// TIA Portal project "ArtecPLC" (V15)

(* hardware
DEVICE "S71500/ET200MP station_1"  S7-1500 station
   slot 0: "Telaio di montaggio_0"  Rack  6ES7 590-1***0-0AA0
   slot 1: "Stazione Principale"  CPU 1515-2 PN  6ES7 515-2AM01-0AB0  V2.5
      slot 3: "Display CPU_1"  6ES7591-1BA00-0AA0
*)

// ===== PLC "Stazione Principale"  CPU 1515-2 PN =====

DATA_BLOCK "DosatoreManuale_DB"   // DB4
{ S7_Optimized_Access := 'TRUE' }
AUTHOR : Valentino-Fabbri
VERSION : 1.14
// stored: InstanceOfName DosatoreManuale
"DosatoreManuale"
BEGIN
END_DATA_BLOCK

// folder: System blocks/Program resources

DATA_BLOCK "ImpulsoEVGas_FB_DosatoreManuale"   // DB1
{ S7_Optimized_Access := 'TRUE' }
AUTHOR : Simatic
FAMILY : IEC
NAME : IEC_TMR
VERSION : 1.0
// stored: InstanceOfName IEC_TIMER
"IEC_TIMER"
BEGIN
END_DATA_BLOCK

DATA_BLOCK "ImpulsoMixer_GasPresente_FB_DosatoreManuale"   // DB2
{ S7_Optimized_Access := 'TRUE' }
AUTHOR : Simatic
FAMILY : IEC
NAME : IEC_TMR
VERSION : 1.0
// stored: InstanceOfName IEC_TIMER
"IEC_TIMER"
BEGIN
END_DATA_BLOCK

DATA_BLOCK "ImpulsoDisco_FB_DosatoreManuale"   // DB3
{ S7_Optimized_Access := 'TRUE' }
AUTHOR : Simatic
FAMILY : IEC
NAME : IEC_TMR
VERSION : 1.0
// stored: InstanceOfName IEC_TIMER
"IEC_TIMER"
BEGIN
END_DATA_BLOCK

// folder: (top level)

FUNCTION_BLOCK "DosatoreManuale"   // FB1, LAD
TITLE = Blocco Dosatore in Manuale
{ S7_Optimized_Access := 'TRUE' }
AUTHOR : Valentino-Fabbri
VERSION : 1.14
   VAR_INPUT
      StopEmergenza : Bool;   // Fornire un bit che se aperto fermi tutto
      GasInPressione : Bool;   // Bit che mi fornisce lo stato del Gas In Pressione
      GasARegime : Bool;   // Bit che mi fornisce lo stato del Gas a Regime
      GasAZero : Bool;   // Bit che mi fornisce lo stato del Gas a zero
      DiscoARegime : Bool;   // Bit che mi fornisce lo stato del Disco a Regime
      DiscoAZero : Bool;   // Bit che mi fornisce lo stato del Disco a zero
      MixerARegime : Bool;   // Bit che mi fornisce lo stato del mixer a Regime
      MixerAZero : Bool;   // Bit che mi fornisce lo stato del mixer a Zero
      DosatoriOkInRicetta : Bool;   // Bit che mi indica se i dosatori sono presenti ed in ricetta
      RicettaMixer : Real;   // Valore fornito dal cliente - misurato in RPM
      RicettaDisco : Real;   // Valore fornito dal cliente - misurato in RPM
      RicettaGas : Real;   // Valore fornito dal cliente - misurato in LPM
      TipoDiAvvio : Bool;   // Modalità di avvio Disco - se prima Disco e poi Mixer, oppure Mixer e poi Disco
   END_VAR
   VAR_OUTPUT
      EVGas : Bool;   // Elettrovalvola Gas Argon
      Mixer : Bool;   // Abilitazione Mixer
      Disco : Bool;   // Abilitazione Disco
      DosatoreAcceso : Bool;   // Flag che indica il dosatore a Regime
   END_VAR
   VAR_IN_OUT
      PulsanteMixerHMI : Bool;   // Pulsante Mixer da HMI
      PulsanteDiscoHMI : Bool;   // Pulsante Disco da HMI
      PulsanteGasHMI : Bool;   // Pulsante Gas da HMI
      PulsanteStopMixer : Bool;   // Stop Mixer da HMI
      PulsanteStopDisco : Bool;   // Stop Disco da HMI
      PulsanteStopGas : Bool;   // Stop Gas da HMI
      ValoreComandoMixer : Real;   // Valore di comando velocità Mixer
      ValoreComandoDisco : Real;   // Valore di comando velocità Disco
      ValoreComandoGas : Real;   // Valore di comando flusso Gas
   END_VAR
   VAR_TEMP
      CondizioniRispettate : Bool;
      "Step" : Array[1..10] of Bool;
      DosatoreSpento : Bool;
      AppoggioPulsanteGas : Bool;
      AppoggioPulsanteMixer : Bool;
      AppoggioPulsanteDisco : Bool;
      AppoggioStopGasDaMixerODisco : Bool;
      AppoggioStopMixerDaDisco : Bool;
      AppoggioStopDiscoDaMixer : Bool;
      StopGas : Bool;
      StopDisco : Bool;
      StopMixer : Bool;
   END_VAR
   VAR_TEMP   // added for the SCL form of the ladder/FBD networks
      _w1 : Bool;
      _w2 : Bool;
      _w3 : Bool;
      _w4 : Bool;
      _w5 : Bool;
      _w6 : Bool;
      _w7 : Bool;
      _w8 : Bool;
      _w9 : Bool;
      _w10 : Bool;
      _w11 : Bool;
      _w12 : Bool;
      _w13 : Bool;
      _w14 : Bool;
   END_VAR
BEGIN

REGION Network 1: Condizioni Iniziali
   // Lo stop di emergenza è un bit che normalmente è chiuso e se aperto vuoldire che una condizione è venuta a mancare in cabina
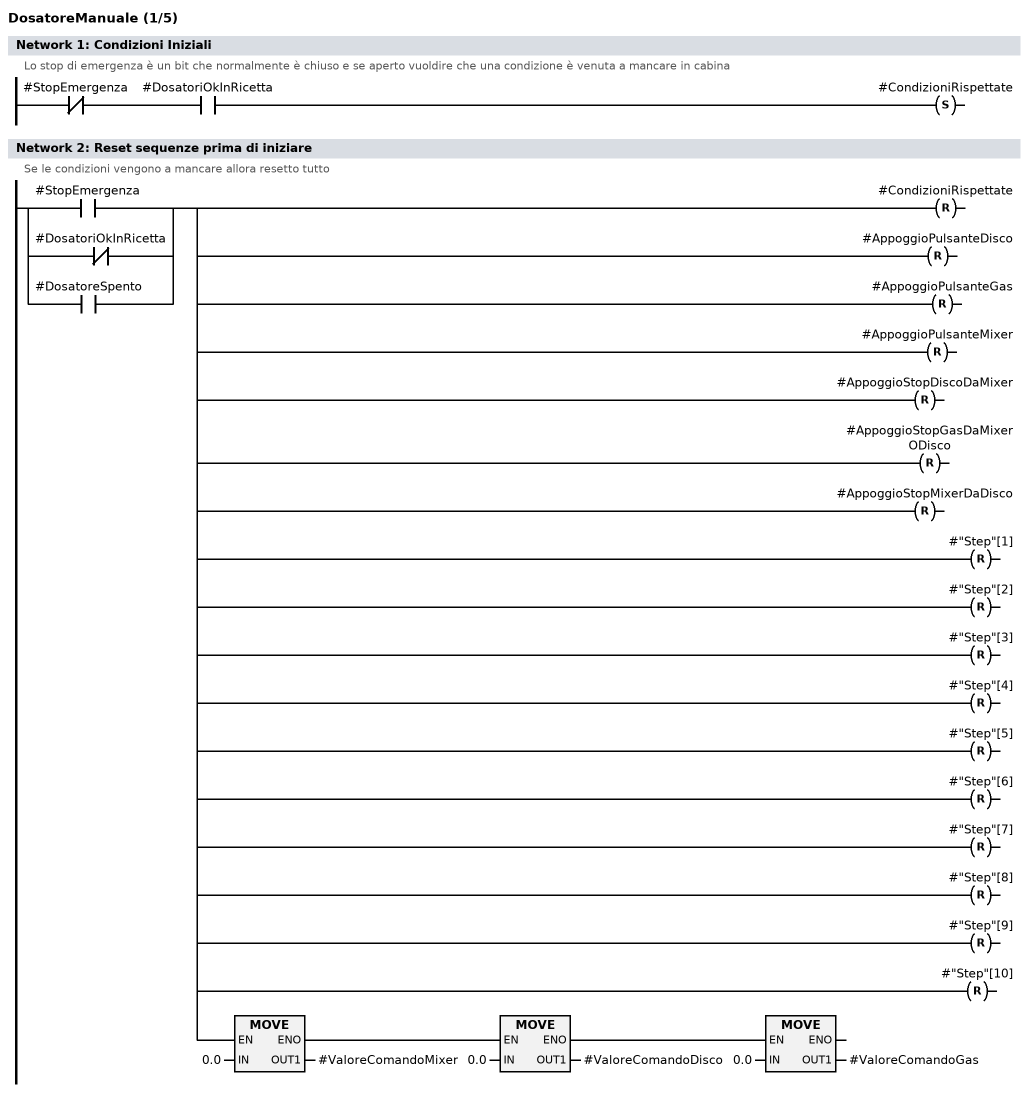
   RUNG wire#powerrail
      I_Contact( #StopEmergenza )
      Contact( #DosatoriOkInRicetta )
      S_Coil( #CondizioniRispettate )
   END_RUNG
   // the same network as SCL:
   IF NOT #StopEmergenza AND #DosatoriOkInRicetta THEN #CondizioniRispettate := TRUE; END_IF;
END_REGION

REGION Network 2: Reset sequenze prima di iniziare
   // Se le condizioni vengono a mancare allora resetto tutto
   RUNG wire#powerrail
      Contact( #StopEmergenza )
      wire#w1
      R_Coil( #CondizioniRispettate )
   END_RUNG
   RUNG wire#powerrail
      I_Contact( #DosatoriOkInRicetta )
   END_RUNG wire#w1
   RUNG wire#powerrail
      Contact( #DosatoreSpento )
   END_RUNG wire#w1
   RUNG wire#w1
      R_Coil( #AppoggioPulsanteDisco )
   END_RUNG
   RUNG wire#w1
      R_Coil( #AppoggioPulsanteGas )
   END_RUNG
   RUNG wire#w1
      R_Coil( #AppoggioPulsanteMixer )
   END_RUNG
   RUNG wire#w1
      R_Coil( #AppoggioStopDiscoDaMixer )
   END_RUNG
   RUNG wire#w1
      R_Coil( #AppoggioStopGasDaMixerODisco )
   END_RUNG
   RUNG wire#w1
      R_Coil( #AppoggioStopMixerDaDisco )
   END_RUNG
   RUNG wire#w1
      R_Coil( #"Step"[1] )
   END_RUNG
   RUNG wire#w1
      R_Coil( #"Step"[2] )
   END_RUNG
   RUNG wire#w1
      R_Coil( #"Step"[3] )
   END_RUNG
   RUNG wire#w1
      R_Coil( #"Step"[4] )
   END_RUNG
   RUNG wire#w1
      R_Coil( #"Step"[5] )
   END_RUNG
   RUNG wire#w1
      R_Coil( #"Step"[6] )
   END_RUNG
   RUNG wire#w1
      R_Coil( #"Step"[7] )
   END_RUNG
   RUNG wire#w1
      R_Coil( #"Step"[8] )
   END_RUNG
   RUNG wire#w1
      R_Coil( #"Step"[9] )
   END_RUNG
   RUNG wire#w1
      R_Coil( #"Step"[10] )
   END_RUNG
   RUNG wire#w1
      Move(in := 0.0, out1 => #ValoreComandoMixer)
      Move(in := 0.0, out1 => #ValoreComandoDisco)
      Move(in := 0.0, out1 => #ValoreComandoGas)
   END_RUNG
   // the same network as SCL:
   IF #StopEmergenza OR NOT #DosatoriOkInRicetta OR #DosatoreSpento THEN
       #CondizioniRispettate := FALSE;
       #AppoggioPulsanteDisco := FALSE;
       #AppoggioPulsanteGas := FALSE;
       #AppoggioPulsanteMixer := FALSE;
       #AppoggioStopDiscoDaMixer := FALSE;
       #AppoggioStopGasDaMixerODisco := FALSE;
       #AppoggioStopMixerDaDisco := FALSE;
       #"Step"[1] := FALSE;
       #"Step"[2] := FALSE;
       #"Step"[3] := FALSE;
       #"Step"[4] := FALSE;
       #"Step"[5] := FALSE;
       #"Step"[6] := FALSE;
       #"Step"[7] := FALSE;
       #"Step"[8] := FALSE;
       #"Step"[9] := FALSE;
       #"Step"[10] := FALSE;
       #ValoreComandoMixer := 0.0;
       #ValoreComandoDisco := 0.0;
       #ValoreComandoGas := 0.0;
   END_IF;
END_REGION

REGION Network 3: Pulsanti di Stop
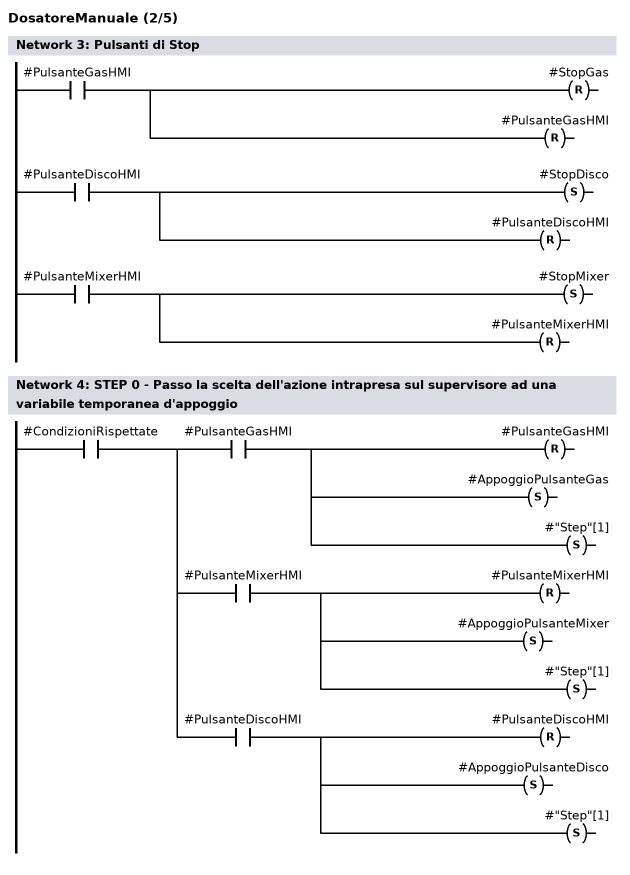
   RUNG wire#powerrail
      Contact( #PulsanteGasHMI )
      wire#w1
      R_Coil( #StopGas )
   END_RUNG
   RUNG wire#w1
      R_Coil( #PulsanteGasHMI )
   END_RUNG
   RUNG wire#powerrail
      Contact( #PulsanteDiscoHMI )
      wire#w2
      S_Coil( #StopDisco )
   END_RUNG
   RUNG wire#w2
      R_Coil( #PulsanteDiscoHMI )
   END_RUNG
   RUNG wire#powerrail
      Contact( #PulsanteMixerHMI )
      wire#w3
      S_Coil( #StopMixer )
   END_RUNG
   RUNG wire#w3
      R_Coil( #PulsanteMixerHMI )
   END_RUNG
   // the same network as SCL:
   IF #PulsanteGasHMI THEN
       #StopGas := FALSE;
       #PulsanteGasHMI := FALSE;
   END_IF;
   IF #PulsanteDiscoHMI THEN
       #StopDisco := TRUE;
       #PulsanteDiscoHMI := FALSE;
   END_IF;
   IF #PulsanteMixerHMI THEN
       #StopMixer := TRUE;
       #PulsanteMixerHMI := FALSE;
   END_IF;
END_REGION

REGION Network 4: STEP 0 - Passo la scelta dell'azione intrapresa sul supervisore ad una variabile temporanea d'appoggio
   RUNG wire#powerrail
      Contact( #CondizioniRispettate )
      wire#w1
      Contact( #PulsanteGasHMI )
      wire#w2
      R_Coil( #PulsanteGasHMI )
   END_RUNG
   RUNG wire#w2
      S_Coil( #AppoggioPulsanteGas )
   END_RUNG
   RUNG wire#w2
      S_Coil( #"Step"[1] )
   END_RUNG
   RUNG wire#w1
      Contact( #PulsanteMixerHMI )
      wire#w3
      R_Coil( #PulsanteMixerHMI )
   END_RUNG
   RUNG wire#w3
      S_Coil( #AppoggioPulsanteMixer )
   END_RUNG
   RUNG wire#w3
      S_Coil( #"Step"[1] )
   END_RUNG
   RUNG wire#w1
      Contact( #PulsanteDiscoHMI )
      wire#w4
      R_Coil( #PulsanteDiscoHMI )
   END_RUNG
   RUNG wire#w4
      S_Coil( #AppoggioPulsanteDisco )
   END_RUNG
   RUNG wire#w4
      S_Coil( #"Step"[1] )
   END_RUNG
   // the same network as SCL:
   #_w1 := #CondizioniRispettate AND #PulsanteGasHMI;
   IF #_w1 THEN
       #PulsanteGasHMI := FALSE;
       #AppoggioPulsanteGas := TRUE;
       #"Step"[1] := TRUE;
   END_IF;
   #_w2 := #CondizioniRispettate AND #PulsanteMixerHMI;
   IF #_w2 THEN
       #PulsanteMixerHMI := FALSE;
       #AppoggioPulsanteMixer := TRUE;
       #"Step"[1] := TRUE;
   END_IF;
   #_w3 := #CondizioniRispettate AND #PulsanteDiscoHMI;
   IF #_w3 THEN
       #PulsanteDiscoHMI := FALSE;
       #AppoggioPulsanteDisco := TRUE;
       #"Step"[1] := TRUE;
   END_IF;
END_REGION

REGION Network 5: STEP 1 - Applico l'azione corrispondente alla scelta effettuata nel segmento precedente
   // Se ho premuto il pulsante GAS - faccio partire solo il GAS
   // Se ho premuto il pulsante Mixer - faccio partire il GAS se non è ancora partito e poi il mixer
   // Se ho premuto il pulsante Disco - faccio partire il GAS , controllo il Tipo Di Avvio, Se Disco-Mixer o Mixer-Disco a seconda di quello partono in rampa il mixer e il disco uno dopo l'altro o viceversa
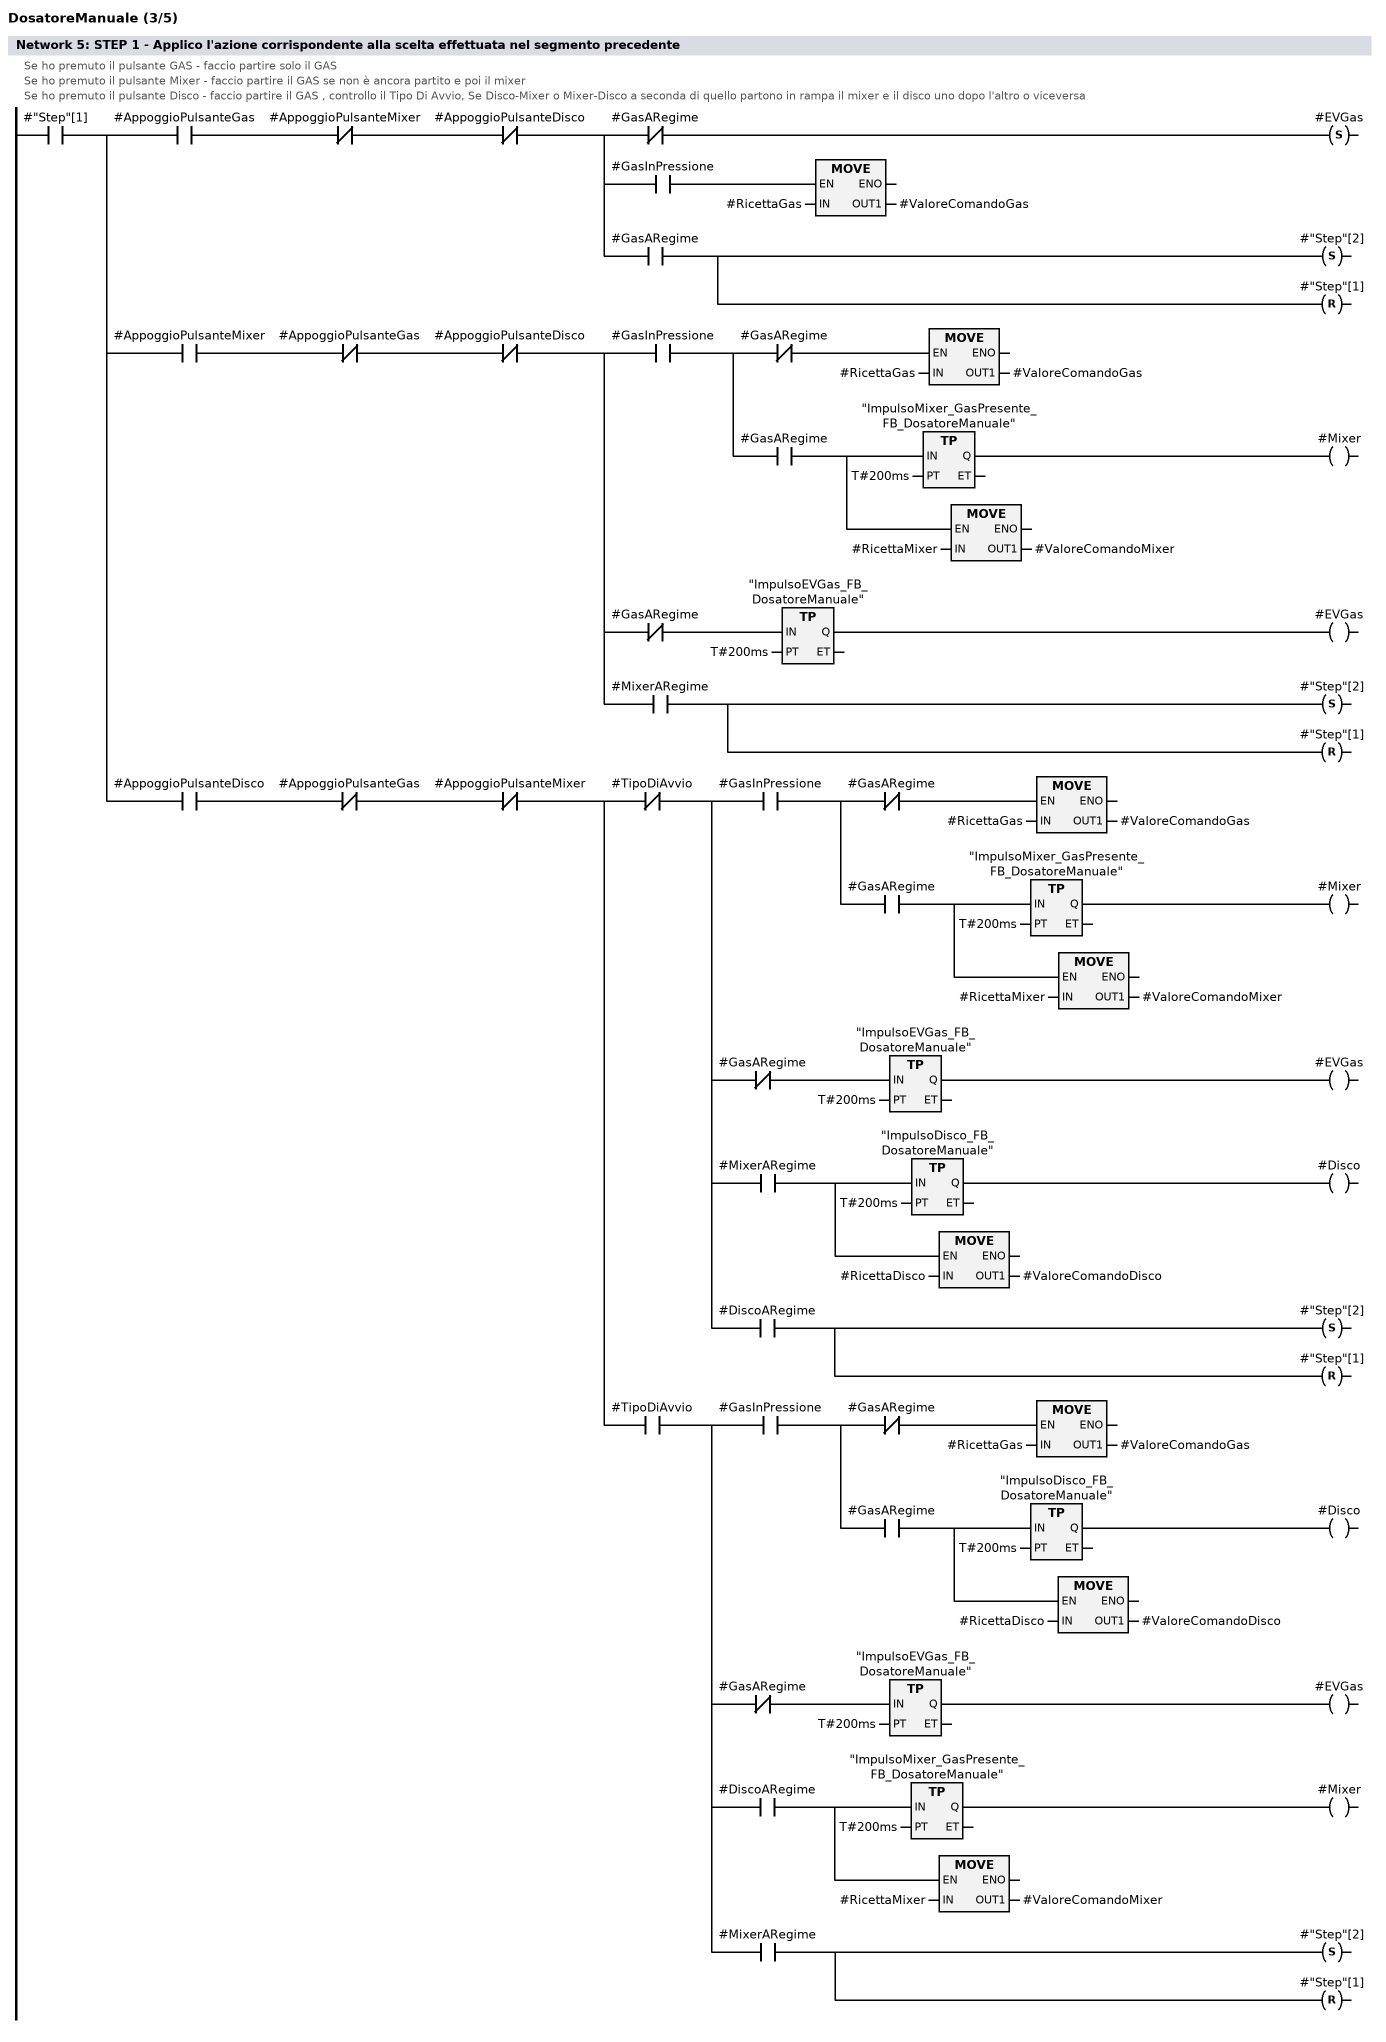
   #_w1 := #"Step"[1] AND #AppoggioPulsanteGas AND NOT #AppoggioPulsanteMixer AND NOT #AppoggioPulsanteDisco;
   IF #_w1 AND NOT #GasARegime THEN #EVGas := TRUE; END_IF;
   IF #_w1 AND #GasInPressione THEN #ValoreComandoGas := #RicettaGas; END_IF;
   #_w2 := #"Step"[1];
   IF #_w1 AND #GasARegime THEN
       #"Step"[2] := TRUE;
       #"Step"[1] := FALSE;
   END_IF;
   #_w3 := #_w2 AND #AppoggioPulsanteMixer AND NOT #AppoggioPulsanteGas AND NOT #AppoggioPulsanteDisco;
   #_w4 := #_w3 AND #GasInPressione;
   IF #_w4 AND NOT #GasARegime THEN #ValoreComandoGas := #RicettaGas; END_IF;
   #_w5 := #_w4 AND #GasARegime;
   "ImpulsoMixer_GasPresente_FB_DosatoreManuale".TP(IN := #_w5, PT := T#200ms);
   #Mixer := "ImpulsoMixer_GasPresente_FB_DosatoreManuale".Q;
   IF #_w5 THEN #ValoreComandoMixer := #RicettaMixer; END_IF;
   "ImpulsoEVGas_FB_DosatoreManuale".TP(IN := #_w3 AND NOT #GasARegime, PT := T#200ms);
   #EVGas := "ImpulsoEVGas_FB_DosatoreManuale".Q;
   IF #_w3 AND #MixerARegime THEN
       #"Step"[2] := TRUE;
       #"Step"[1] := FALSE;
   END_IF;
   #_w6 := #_w2 AND #AppoggioPulsanteDisco AND NOT #AppoggioPulsanteGas AND NOT #AppoggioPulsanteMixer;
   #_w7 := #_w6 AND NOT #TipoDiAvvio;
   #_w8 := #_w7 AND #GasInPressione;
   IF #_w8 AND NOT #GasARegime THEN #ValoreComandoGas := #RicettaGas; END_IF;
   #_w9 := #_w8 AND #GasARegime;
   "ImpulsoMixer_GasPresente_FB_DosatoreManuale".TP(IN := #_w9, PT := T#200ms);
   #Mixer := "ImpulsoMixer_GasPresente_FB_DosatoreManuale".Q;
   IF #_w9 THEN #ValoreComandoMixer := #RicettaMixer; END_IF;
   "ImpulsoEVGas_FB_DosatoreManuale".TP(IN := #_w7 AND NOT #GasARegime, PT := T#200ms);
   #EVGas := "ImpulsoEVGas_FB_DosatoreManuale".Q;
   #_w10 := #_w7 AND #MixerARegime;
   "ImpulsoDisco_FB_DosatoreManuale".TP(IN := #_w10, PT := T#200ms);
   #Disco := "ImpulsoDisco_FB_DosatoreManuale".Q;
   IF #_w10 THEN #ValoreComandoDisco := #RicettaDisco; END_IF;
   IF #_w7 AND #DiscoARegime THEN
       #"Step"[2] := TRUE;
       #"Step"[1] := FALSE;
   END_IF;
   #_w11 := #_w6 AND #TipoDiAvvio;
   #_w12 := #_w11 AND #GasInPressione;
   IF #_w12 AND NOT #GasARegime THEN #ValoreComandoGas := #RicettaGas; END_IF;
   #_w13 := #_w12 AND #GasARegime;
   "ImpulsoDisco_FB_DosatoreManuale".TP(IN := #_w13, PT := T#200ms);
   #Disco := "ImpulsoDisco_FB_DosatoreManuale".Q;
   IF #_w13 THEN #ValoreComandoDisco := #RicettaDisco; END_IF;
   "ImpulsoEVGas_FB_DosatoreManuale".TP(IN := #_w11 AND NOT #GasARegime, PT := T#200ms);
   #EVGas := "ImpulsoEVGas_FB_DosatoreManuale".Q;
   #_w14 := #_w11 AND #DiscoARegime;
   "ImpulsoMixer_GasPresente_FB_DosatoreManuale".TP(IN := #_w14, PT := T#200ms);
   #Mixer := "ImpulsoMixer_GasPresente_FB_DosatoreManuale".Q;
   IF #_w14 THEN #ValoreComandoMixer := #RicettaMixer; END_IF;
   IF #_w11 AND #MixerARegime THEN
       #"Step"[2] := TRUE;
       #"Step"[1] := FALSE;
   END_IF;
END_REGION

REGION Network 6: STEP 2 - Spegnimento Gas o Mixer e poi Gas
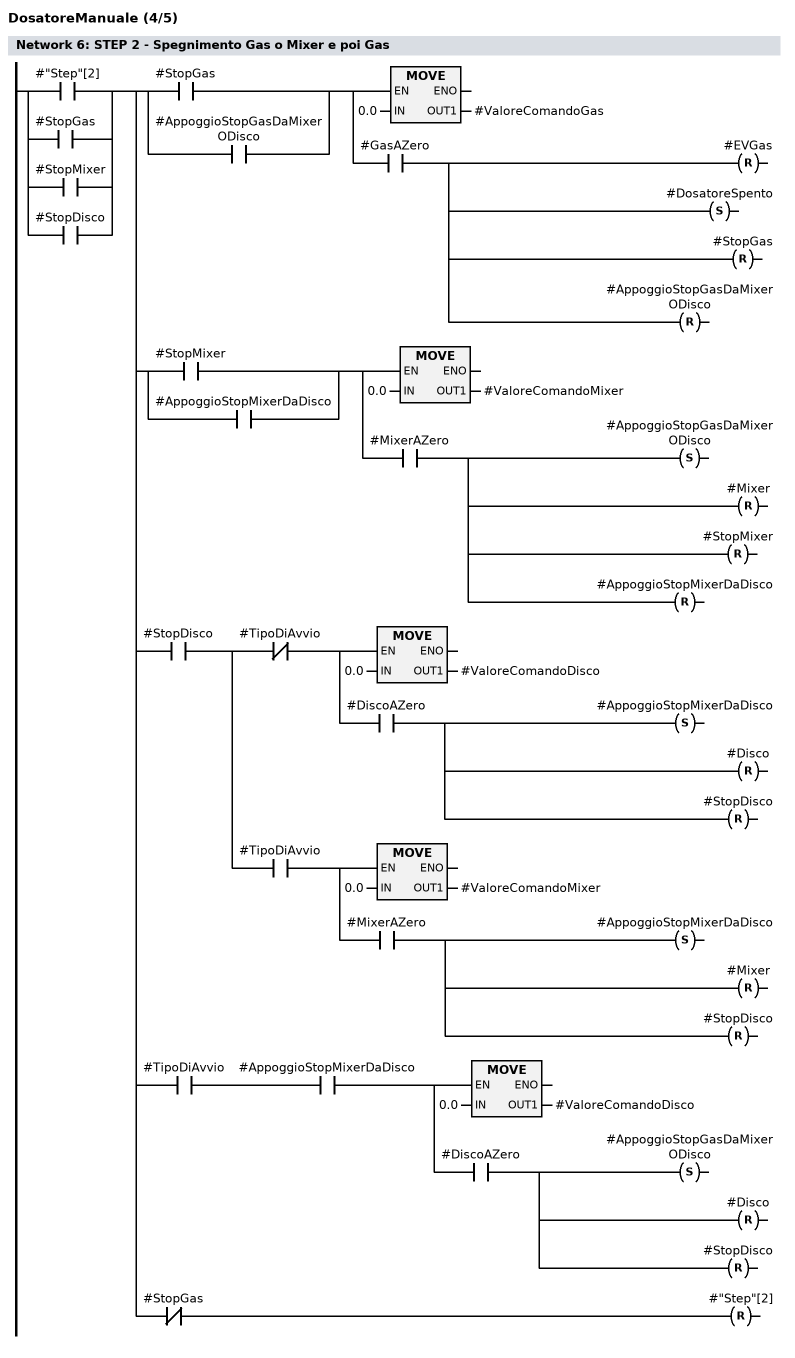
   RUNG wire#powerrail
      Contact( #"Step"[2] )
      wire#w1
      Contact( #StopGas )
      wire#w2
      Move(in := 0.0, out1 => #ValoreComandoGas)
   END_RUNG
   RUNG wire#powerrail
      Contact( #StopGas )
   END_RUNG wire#w1
   RUNG wire#powerrail
      Contact( #StopMixer )
   END_RUNG wire#w1
   RUNG wire#powerrail
      Contact( #StopDisco )
   END_RUNG wire#w1
   RUNG wire#w1
      Contact( #AppoggioStopGasDaMixerODisco )
   END_RUNG wire#w2
   RUNG wire#w2
      Contact( #GasAZero )
      wire#w3
      R_Coil( #EVGas )
   END_RUNG
   RUNG wire#w3
      S_Coil( #DosatoreSpento )
   END_RUNG
   RUNG wire#w3
      R_Coil( #StopGas )
   END_RUNG
   RUNG wire#w3
      R_Coil( #AppoggioStopGasDaMixerODisco )
   END_RUNG
   RUNG wire#w1
      Contact( #StopMixer )
      wire#w4
      Move(in := 0.0, out1 => #ValoreComandoMixer)
   END_RUNG
   RUNG wire#w1
      Contact( #AppoggioStopMixerDaDisco )
   END_RUNG wire#w4
   RUNG wire#w4
      Contact( #MixerAZero )
      wire#w5
      S_Coil( #AppoggioStopGasDaMixerODisco )
   END_RUNG
   RUNG wire#w5
      R_Coil( #Mixer )
   END_RUNG
   RUNG wire#w5
      R_Coil( #StopMixer )
   END_RUNG
   RUNG wire#w5
      R_Coil( #AppoggioStopMixerDaDisco )
   END_RUNG
   RUNG wire#w1
      Contact( #StopDisco )
      wire#w6
      I_Contact( #TipoDiAvvio )
      wire#w7
      Move(in := 0.0, out1 => #ValoreComandoDisco)
   END_RUNG
   RUNG wire#w7
      Contact( #DiscoAZero )
      wire#w8
      S_Coil( #AppoggioStopMixerDaDisco )
   END_RUNG
   RUNG wire#w8
      R_Coil( #Disco )
   END_RUNG
   RUNG wire#w8
      R_Coil( #StopDisco )
   END_RUNG
   RUNG wire#w6
      Contact( #TipoDiAvvio )
      wire#w9
      Move(in := 0.0, out1 => #ValoreComandoMixer)
   END_RUNG
   RUNG wire#w9
      Contact( #MixerAZero )
      wire#w10
      S_Coil( #AppoggioStopMixerDaDisco )
   END_RUNG
   RUNG wire#w10
      R_Coil( #Mixer )
   END_RUNG
   RUNG wire#w10
      R_Coil( #StopDisco )
   END_RUNG
   RUNG wire#w1
      Contact( #TipoDiAvvio )
      Contact( #AppoggioStopMixerDaDisco )
      wire#w11
      Move(in := 0.0, out1 => #ValoreComandoDisco)
   END_RUNG
   RUNG wire#w11
      Contact( #DiscoAZero )
      wire#w12
      S_Coil( #AppoggioStopGasDaMixerODisco )
   END_RUNG
   RUNG wire#w12
      R_Coil( #Disco )
   END_RUNG
   RUNG wire#w12
      R_Coil( #StopDisco )
   END_RUNG
   RUNG wire#w1
      I_Contact( #StopGas )
      R_Coil( #"Step"[2] )
   END_RUNG
   // the same network as SCL:
   #_w1 := #"Step"[2] OR #StopGas OR #StopMixer OR #StopDisco;
   #_w2 := #_w1 AND (#StopGas OR #AppoggioStopGasDaMixerODisco);
   IF #_w2 THEN #ValoreComandoGas := 0.0; END_IF;
   IF #_w2 AND #GasAZero THEN
       #EVGas := FALSE;
       #DosatoreSpento := TRUE;
       #StopGas := FALSE;
       #AppoggioStopGasDaMixerODisco := FALSE;
   END_IF;
   #_w3 := #_w1 AND (#StopMixer OR #AppoggioStopMixerDaDisco);
   IF #_w3 THEN #ValoreComandoMixer := 0.0; END_IF;
   IF #_w3 AND #MixerAZero THEN
       #AppoggioStopGasDaMixerODisco := TRUE;
       #Mixer := FALSE;
       #StopMixer := FALSE;
       #AppoggioStopMixerDaDisco := FALSE;
   END_IF;
   #_w4 := #_w1 AND #StopDisco;
   #_w5 := #_w4 AND NOT #TipoDiAvvio;
   IF #_w5 THEN #ValoreComandoDisco := 0.0; END_IF;
   IF #_w5 AND #DiscoAZero THEN
       #AppoggioStopMixerDaDisco := TRUE;
       #Disco := FALSE;
       #StopDisco := FALSE;
   END_IF;
   #_w6 := #_w4 AND #TipoDiAvvio;
   IF #_w6 THEN #ValoreComandoMixer := 0.0; END_IF;
   IF #_w6 AND #MixerAZero THEN
       #AppoggioStopMixerDaDisco := TRUE;
       #Mixer := FALSE;
       #StopDisco := FALSE;
   END_IF;
   #_w7 := #_w1 AND #TipoDiAvvio AND #AppoggioStopMixerDaDisco;
   IF #_w7 THEN #ValoreComandoDisco := 0.0; END_IF;
   IF #_w7 AND #DiscoAZero THEN
       #AppoggioStopGasDaMixerODisco := TRUE;
       #Disco := FALSE;
       #StopDisco := FALSE;
   END_IF;
   IF #_w1 AND NOT #StopGas THEN #"Step"[2] := FALSE; END_IF;
END_REGION

REGION Network 7: Flag per dosatore avviato
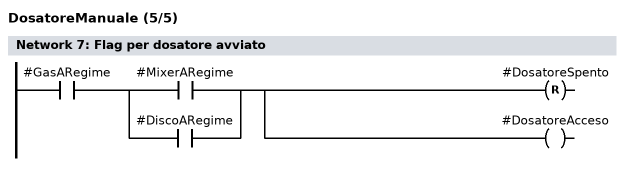
   RUNG wire#powerrail
      Contact( #GasARegime )
      wire#w1
      Contact( #MixerARegime )
      wire#w2
      R_Coil( #DosatoreSpento )
   END_RUNG
   RUNG wire#w1
      Contact( #DiscoARegime )
   END_RUNG wire#w2
   RUNG wire#w2
      Coil( #DosatoreAcceso )
   END_RUNG
   // the same network as SCL:
   #_w1 := #GasARegime AND (#MixerARegime OR #DiscoARegime);
   IF #_w1 THEN #DosatoreSpento := FALSE; END_IF;
   #DosatoreAcceso := #_w1;
END_REGION
END_FUNCTION_BLOCK

ORGANIZATION_BLOCK "Main"   // OB1, LAD, ProgramCycle
TITLE = "Main Program Sweep (Cycle)"
{ S7_Optimized_Access := 'TRUE' }
VERSION : 0.1
   VAR_INPUT
      Initial_Call : Bool;   // Initial call of this OB
      Remanence : Bool;   // =True, if remanent data are available
   END_VAR
BEGIN

REGION Network 1: DOSATORE 1 in Manuale
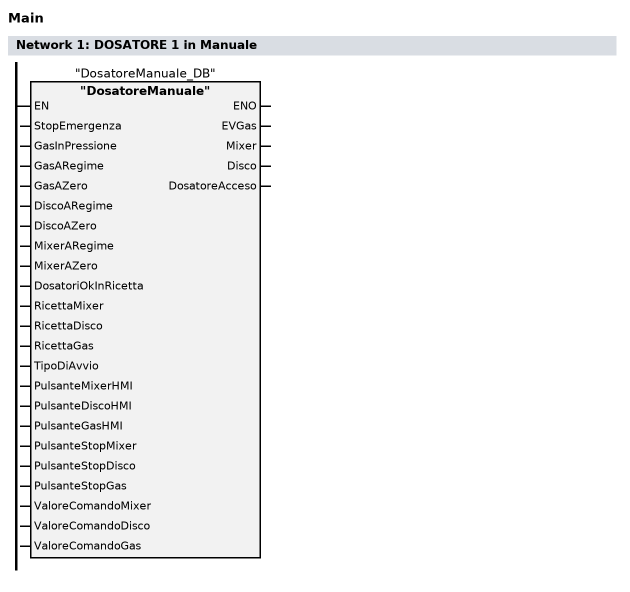
   RUNG wire#powerrail
      "DosatoreManuale_DB"(StopEmergenza :=, GasInPressione :=, GasARegime :=, GasAZero :=, DiscoARegime :=, DiscoAZero :=, MixerARegime :=, MixerAZero :=, DosatoriOkInRicetta :=, RicettaMixer :=, RicettaDisco :=, RicettaGas :=, TipoDiAvvio :=, PulsanteMixerHMI :=, PulsanteDiscoHMI :=, PulsanteGasHMI :=, PulsanteStopMixer :=, PulsanteStopDisco :=, PulsanteStopGas :=, ValoreComandoMixer :=, ValoreComandoDisco :=, ValoreComandoGas :=, EVGas =>, Mixer =>, Disco =>, DosatoreAcceso =>)
   END_RUNG
   // the same network as SCL:
   "DosatoreManuale_DB"();   // "DosatoreManuale"
END_REGION
END_ORGANIZATION_BLOCK